{attribute addProperty BoxType "EK1100-0000-0018"}
{attribute addProperty Id "Beckhoff_ER6xxxEK1122Beckhoff_ER6xxxEK1122_6F47836B3568446"}
{attribute addProperty CRC "2565096126"}
{attribute addProperty SizeInBites "3568"}
{attribute addProperty SizeInBytes "446"}
TYPE Beckhoff_ER6xxx_98E442BE EXTENDS EK1100_179A0949 :
STRUCT
	{attribute addProperty Name "Beckhoff_ER6xxxEK1122"}
	Beckhoff_ER6xxxEK1122 : Beckhoff_ER6xxxEK1122_6F47836B;
END_STRUCT
END_TYPE

(* stored: Version 1.2.0.0, ProductVersion 3.1.4024.9
   DUT Beckhoff_ER6xxx_98E442BE: Id {3d4ea4a1-6bc3-4e98-a7ef-d1cf01151711} *)
